{attribute addProperty BoxType "EL9560-0000-0016"}
{attribute addProperty Id "Power_OKAT %I*BOOL81"}
{attribute addProperty CRC "843727106"}
{attribute addProperty SizeInBites "8"}
{attribute addProperty SizeInBytes "1"}
TYPE Status_Uo_324A4102 :
STRUCT
	{attribute addProperty Name "Power_OK"}
	Power_OK AT %I* : BOOL;
END_STRUCT
END_TYPE

(* stored: Version 1.2.0.0, ProductVersion 3.1.4024.9
   DUT Status_Uo_324A4102: Id {d38dc71d-9e17-4d34-b740-b239dc01ca4b} *)
